FUNCTION_BLOCK FB_Reset
VAR_IN_OUT
	stAxis 	 	: ARRAY [GVL.cXP .. GVL.cXM] OF ST_AxisGroup;	
	bResetting	: BOOL;
	bResetEntry : BOOL;
END_VAR
VAR
	nCurrentState 	: INT;
	nNextState		: INT := 100;
	//a,b,c,d,e : INT;
	fbResetTimer	: TON ;
END_VAR

IF bResetEntry THEN
	nNextState := 50;
	bResetEntry := FALSE;
END_IF

nCurrentState := nNextState;
CASE nCurrentstate OF
	
	50:
		stAxis[GVL.cXP].mcReset(axis:=stAxis[GVL.cXP].axisRef, Execute:=TRUE);
		stAxis[GVL.cXM].mcReset(axis:=stAxis[GVL.cXM].axisRef, Execute:=TRUE);
		IF stAxis[GVL.cXP].mcReset.Done AND stAxis[GVL.cXM].mcReset.Done THEN
			stAxis[GVL.cXP].mcReset(axis:=stAxis[GVL.cXP].axisRef, Execute:=FALSE);
			stAxis[GVL.cXM].mcReset(axis:=stAxis[GVL.cXM].axisRef, Execute:=FALSE);
			nNextState := 100;
		END_IF
		//e := e+1;
		
	100:
		stAxis[GVL.cXP].mcStop(Axis:=stAxis[GVL.cXP].axisRef, Execute:=FALSE);
		stAxis[GVL.cXM].mcStop(Axis:=stAxis[GVL.cXM].axisRef, Execute:=FALSE);
		fbResetTimer(IN:=TRUE, PT:=T#100MS);
		IF FBResetTimer.Q THEN
			fbResetTimer(IN:=FALSE);
			nNextState:=200;
		END_IF
		//nNextState := 200;
		//a := a+1;
		
	200:
		stAxis[GVL.cXP].mcStop(Axis:=stAxis[GVL.cXP].axisRef, Execute:=TRUE);
		stAxis[GVL.cXM].mcStop(Axis:=stAxis[GVL.cXM].axisRef, Execute:=TRUE);
		IF stAxis[GVL.cXP].mcStop.Done AND stAxis[GVL.cXM].mcStop.Done THEN 
			stAxis[GVL.cXP].mcStop(Axis:=stAxis[GVL.cXP].axisRef, Execute:=FALSE);
			stAxis[GVL.cXM].mcStop(Axis:=stAxis[GVL.cXM].axisRef, Execute:=FALSE);
			nNextState := 300;
			//b := b+1;
		END_IF
		//c := c+1;
	
	300:
		stAxis[GVL.cXP].mcMoveAbs(Axis:=stAxis[GVL.cXP].axisRef, Execute:=FALSE);
		stAxis[GVL.cXM].mcMoveAbs(Axis:=stAxis[GVL.cXM].axisRef, Execute:=FALSE);
		stAxis[GVL.cXP].mcMoveRel(Axis:=stAxis[GVL.cXP].axisRef, Execute:=FALSE);
		stAxis[GVL.cXM].mcMoveRel(Axis:=stAxis[GVL.cXM].axisRef, Execute:=FALSE);
		stAxis[GVL.cXP].mcJog(Axis:=stAxis[GVL.cXP].axisRef, JogForward:=FALSE, JogBackwards:=FALSE);
		stAxis[GVL.cXM].mcJog(Axis:=stAxis[GVL.cXM].axisRef, JogForward:=FALSE, JogBackwards:=FALSE);
		nNextState := 400;
		
	400:
		stAxis[GVL.cXP].mcReset(axis:=stAxis[GVL.cXP].axisRef, Execute:=TRUE);
		stAxis[GVL.cXM].mcReset(axis:=stAxis[GVL.cXM].axisRef, Execute:=TRUE);
		IF stAxis[GVL.cXP].mcReset.Done AND stAxis[GVL.cXM].mcReset.Done THEN
			stAxis[GVL.cXP].mcReset(axis:=stAxis[GVL.cXP].axisRef, Execute:=FALSE);
			stAxis[GVL.cXM].mcReset(axis:=stAxis[GVL.cXM].axisRef, Execute:=FALSE);
			bResetting := FALSE;
			nNextState := 100;
		END_IF
		//d := d+1;

END_CASE

END_FUNCTION_BLOCK

(* stored: Version 1.1.0.1, ProductVersion 3.1.4024.3
   POU FB_Reset: Id {899b01f2-f2a5-415e-96f0-f718ca072402}, SpecialFunc None *)
